// TIA Portal V21 export
DATA_BLOCK "Ai_Faceplate_Db"   // DB107
{ S7_Optimized_Access := 'TRUE' }
// stored: AutoNumber false, MemoryReserve 100
   VAR
      Ai01 : "Ai_Faceplate";   // Ticr01NfcoLineTemp
      Ai02 : "Ai_Faceplate";   // Ticr02VfcoLineTemp
      Ai03 : "Ai_Faceplate";   // Ticr03SvcoLineTemp
      Ai04 : "Ai_Faceplate";   // Ticr04VdcoTemp
      Ai05 : "Ai_Faceplate";   // Ticr05CipPumpDrainTemp
      Ai06 : "Ai_Faceplate";   // Ticr06Pf01InLineTemp
      Ai07 : "Ai_Faceplate";   // Ticr07Pf02InLineTemp
      Ai08 : "Ai_Faceplate";   // Ticr08Pf02OutLineTemp
      Ai09 : "Ai_Faceplate";   // Ticr09PtlDrainTemp
      Ai10 : "Ai_Faceplate";   // Ticr10VesselTemp
      Ai11 : "Ai_Faceplate";   // Picr01VesselPressure
      Ai12 : "Ai_Faceplate";   // Picr02VesselRclLine
      Ai13 : "Ai_Faceplate";   // Picr03Pf01OutLinePressure
      Ai14 : "Ai_Faceplate";   // Picr04Pf02OutLinePressure
      Ai15 : "Ai_Faceplate";   // Cicr01ProcessDrainConductivity
      Ai16 : "Ai_Faceplate";   // AiSpare1
      Ai17 : "Ai_Faceplate";   // AiSpare2
      Ai18 : "Ai_Faceplate";   // AiSpare3
      Ai19 : "Ai_Faceplate";   // AiSpare4
      Ai20 : "Ai_Faceplate";   // AiSpare5
      Ai21 : "Ai_Faceplate";   // AiSpare6
      Ai22 : "Ai_Faceplate";   // AiSpare7
      Ai23 : "Ai_Faceplate";   // AiSpare8
      Ai24 : "Ai_Faceplate";   // AiSpare9
      Ai25 : "Ai_Faceplate";
      Ai26 : "Ai_Faceplate";
   END_VAR
BEGIN
END_DATA_BLOCK
